TYPE ST_RecCmd ://纠偏系统
STRUCT
    bLock:				BOOL;	//纠偏外部锁定
	bAuto:				BOOL;	//纠偏自动
	bManual:           BOOL;  //纠偏手动
	bCentre:           BOOL;	//纠偏居中

END_STRUCT
END_TYPE

(* stored: Version 1.1.0.1, ProductVersion 3.1.4024.9
   DUT ST_RecCmd: Id {3e6fa4ba-bed9-4a1c-b570-830a3e55392d} *)
